# EPICS IOC start-up script: iocsh/epi8600-eth-ctrl.iocsh
#- ###         MODBUS   epi8600   iocsh             ###
#- ####################################################
#- >> Mandatory
#- ASYN_PORT_NAME - MODBUS ASYN <name>
#- IP_ADDR	  - ethernet address
#- IOCNAME	  - Prefix for the asynRec
#-
#- >> Optional
#- IP_PORT	  - IP port number, default 502
#- TIME_OUT	  - Modbus time-out, default 1900 ms
#- WRITE_DELAY	  - Modbus write delay, default 500 ms

addScan(60)

#-https://epics-modules.github.io/master/asyn/R4-42/asynDriver.html
#-Specify the TCP endpoint and give your 'bus' an arbitrary name eg. "asynstream1".
#- drvAsynIPPortConfigure( portName,
#- 			   hostInfo,
#-			   priority,
#-			   noAutoConnect,
#-			   noProcessEos)
#
drvAsynIPPortConfigure("$(ASYN_PORT_NAME)","$(IP_ADDR):$(IP_PORT=502)",0,0,1)

#modbusInterposeConfig(portName,
#                      linkType,
#                      timeoutMsec,
#                      writeDelayMsec)

modbusInterposeConfig("$(ASYN_PORT_NAME)",0,$(TIME_OUT=1900),$(WRITE_DELAY=500))

asynSetTraceIOMask "$(ASYN_PORT_NAME)",0,4   # Enable traceIOHex
#asynSetTraceMask "$(ASYN_PORT_NAME)",0,9     # Enable traceError and traceIODriver
